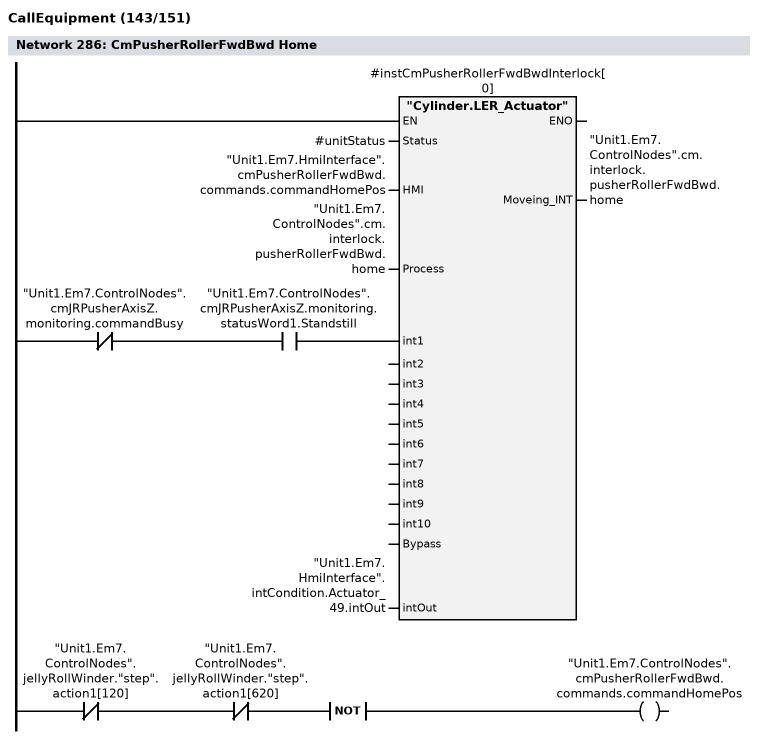
   RUNG wire#powerrail
      #instCmPusherRollerFwdBwdInterlock[0](int1 := wire#w1, Status := #unitStatus, HMI := "Unit1.Em7.HmiInterface".cmPusherRollerFwdBwd.commands.commandHomePos, Process := "Unit1.Em7.ControlNodes".cm.interlock.pusherRollerFwdBwd.home, int2 :=, int3 :=, int4 :=, int5 :=, int6 :=, int7 :=, int8 :=, int9 :=, int10 :=, Bypass :=, intOut := "Unit1.Em7.HmiInterface".intCondition.Actuator_49.intOut, Moveing_INT => "Unit1.Em7.ControlNodes".cm.interlock.pusherRollerFwdBwd.home)
   END_RUNG
   RUNG wire#powerrail
      I_Contact( "Unit1.Em7.ControlNodes".cmJRPusherAxisZ.monitoring.commandBusy )
      Contact( "Unit1.Em7.ControlNodes".cmJRPusherAxisZ.monitoring.statusWord1.Standstill )
   END_RUNG wire#w1
   RUNG wire#powerrail
      I_Contact( "Unit1.Em7.ControlNodes".jellyRollWinder."step".action1[120] )
      I_Contact( "Unit1.Em7.ControlNodes".jellyRollWinder."step".action1[620] )
      Not()
      Coil( "Unit1.Em7.ControlNodes".cmPusherRollerFwdBwd.commands.commandHomePos )
   END_RUNG
   // the same network as SCL:
   #instCmPusherRollerFwdBwdInterlock[0](Status := #unitStatus,   // "Cylinder.LER_Actuator"
                           HMI := "Unit1.Em7.HmiInterface".cmPusherRollerFwdBwd.commands.commandHomePos,
                           Process := "Unit1.Em7.ControlNodes".cm.interlock.pusherRollerFwdBwd.home,
                           int1 := NOT "Unit1.Em7.ControlNodes".cmJRPusherAxisZ.monitoring.commandBusy AND "Unit1.Em7.ControlNodes".cmJRPusherAxisZ.monitoring.statusWord1.Standstill,
                           intOut := "Unit1.Em7.HmiInterface".intCondition.Actuator_49.intOut,
                           Moveing_INT => "Unit1.Em7.ControlNodes".cm.interlock.pusherRollerFwdBwd.home);
   "Unit1.Em7.ControlNodes".cmPusherRollerFwdBwd.commands.commandHomePos := NOT (NOT "Unit1.Em7.ControlNodes".jellyRollWinder."step".action1[120] AND NOT "Unit1.Em7.ControlNodes".jellyRollWinder."step".action1[620]);
END_REGION

REGION Network 287: CmPusherRollerFwdBwd Work
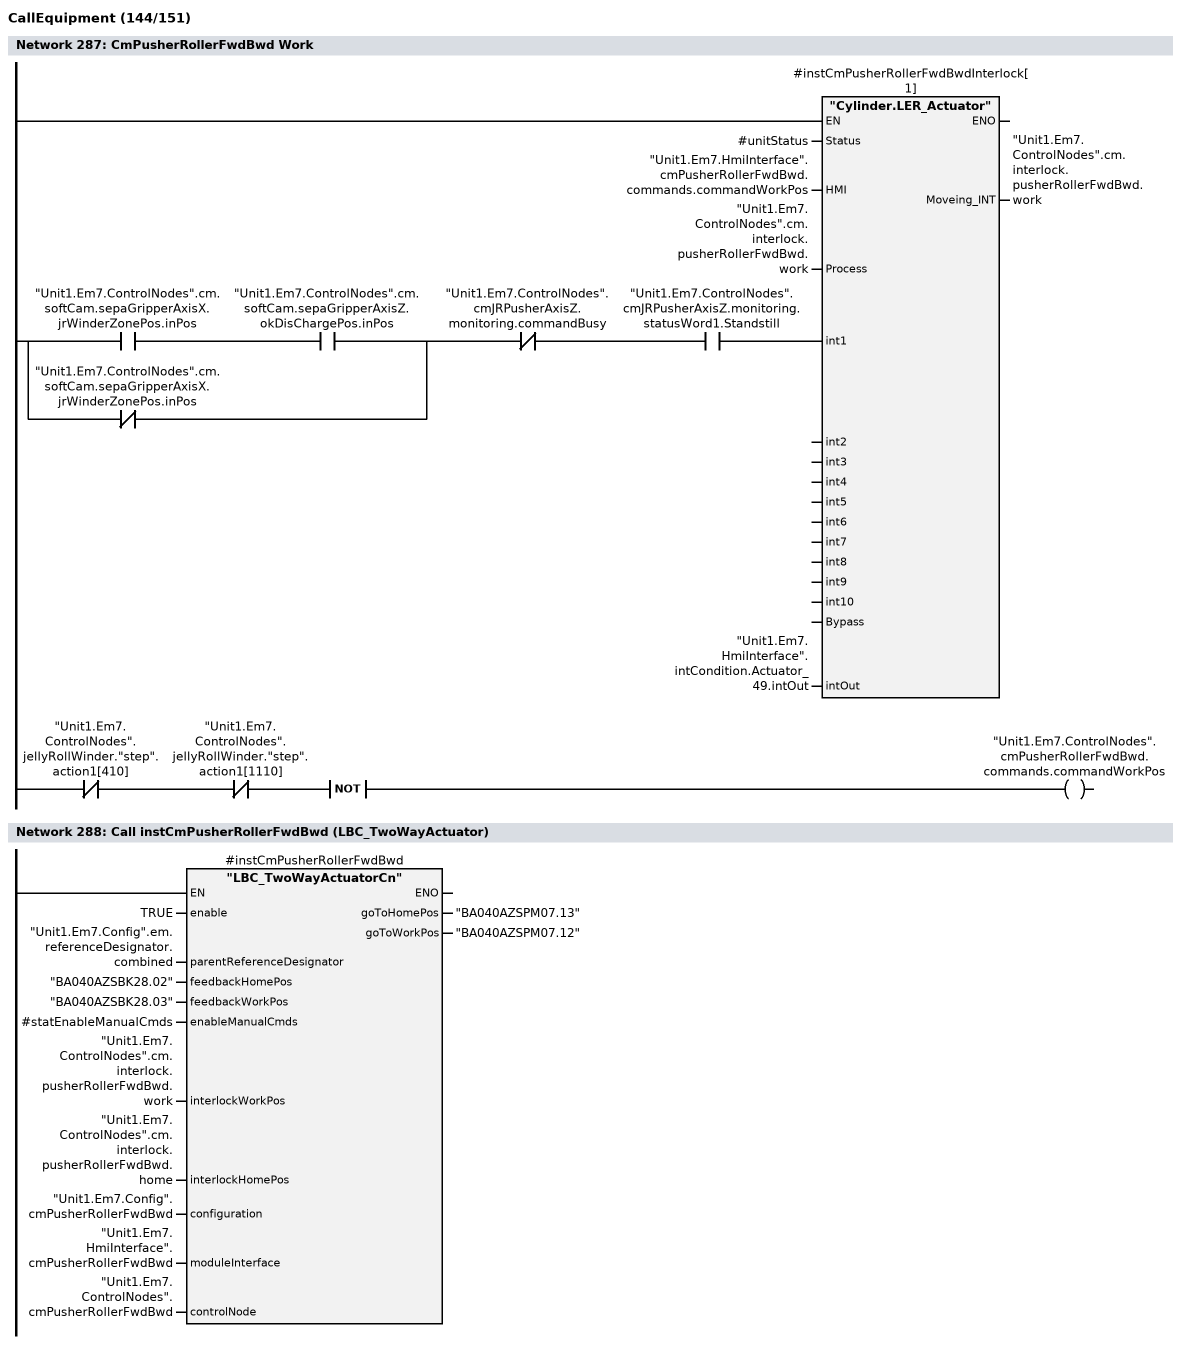
   RUNG wire#powerrail
      #instCmPusherRollerFwdBwdInterlock[1](int1 := wire#w2, Status := #unitStatus, HMI := "Unit1.Em7.HmiInterface".cmPusherRollerFwdBwd.commands.commandWorkPos, Process := "Unit1.Em7.ControlNodes".cm.interlock.pusherRollerFwdBwd.work, int2 :=, int3 :=, int4 :=, int5 :=, int6 :=, int7 :=, int8 :=, int9 :=, int10 :=, Bypass :=, intOut := "Unit1.Em7.HmiInterface".intCondition.Actuator_49.intOut, Moveing_INT => "Unit1.Em7.ControlNodes".cm.interlock.pusherRollerFwdBwd.work)
   END_RUNG
   RUNG wire#powerrail
      Contact( "Unit1.Em7.ControlNodes".cm.softCam.sepaGripperAxisX.jrWinderZonePos.inPos )
      Contact( "Unit1.Em7.ControlNodes".cm.softCam.sepaGripperAxisZ.okDisChargePos.inPos )
      wire#w1
      I_Contact( "Unit1.Em7.ControlNodes".cmJRPusherAxisZ.monitoring.commandBusy )
      Contact( "Unit1.Em7.ControlNodes".cmJRPusherAxisZ.monitoring.statusWord1.Standstill )
   END_RUNG wire#w2
   RUNG wire#powerrail
      I_Contact( "Unit1.Em7.ControlNodes".cm.softCam.sepaGripperAxisX.jrWinderZonePos.inPos )
   END_RUNG wire#w1
   RUNG wire#powerrail
      I_Contact( "Unit1.Em7.ControlNodes".jellyRollWinder."step".action1[410] )
      I_Contact( "Unit1.Em7.ControlNodes".jellyRollWinder."step".action1[1110] )
      Not()
      Coil( "Unit1.Em7.ControlNodes".cmPusherRollerFwdBwd.commands.commandWorkPos )
   END_RUNG
   // the same network as SCL:
   #instCmPusherRollerFwdBwdInterlock[1](Status := #unitStatus,   // "Cylinder.LER_Actuator"
                           HMI := "Unit1.Em7.HmiInterface".cmPusherRollerFwdBwd.commands.commandWorkPos,
                           Process := "Unit1.Em7.ControlNodes".cm.interlock.pusherRollerFwdBwd.work,
                           int1 := (("Unit1.Em7.ControlNodes".cm.softCam.sepaGripperAxisX.jrWinderZonePos.inPos AND "Unit1.Em7.ControlNodes".cm.softCam.sepaGripperAxisZ.okDisChargePos.inPos) OR NOT "Unit1.Em7.ControlNodes".cm.softCam.sepaGripperAxisX.jrWinderZonePos.inPos) AND NOT "Unit1.Em7.ControlNodes".cmJRPusherAxisZ.monitoring.commandBusy AND "Unit1.Em7.ControlNodes".cmJRPusherAxisZ.monitoring.statusWord1.Standstill,
                           intOut := "Unit1.Em7.HmiInterface".intCondition.Actuator_49.intOut,
                           Moveing_INT => "Unit1.Em7.ControlNodes".cm.interlock.pusherRollerFwdBwd.work);
   "Unit1.Em7.ControlNodes".cmPusherRollerFwdBwd.commands.commandWorkPos := NOT (NOT "Unit1.Em7.ControlNodes".jellyRollWinder."step".action1[410] AND NOT "Unit1.Em7.ControlNodes".jellyRollWinder."step".action1[1110]);
END_REGION

REGION Network 288: Call instCmPusherRollerFwdBwd (LBC_TwoWayActuator)
   RUNG wire#powerrail
      #instCmPusherRollerFwdBwd(enable := TRUE, parentReferenceDesignator := "Unit1.Em7.Config".em.referenceDesignator.combined, feedbackHomePos := "BA040AZSBK28.02", feedbackWorkPos := "BA040AZSBK28.03", enableManualCmds := #statEnableManualCmds, interlockWorkPos := "Unit1.Em7.ControlNodes".cm.interlock.pusherRollerFwdBwd.work, interlockHomePos := "Unit1.Em7.ControlNodes".cm.interlock.pusherRollerFwdBwd.home, configuration := "Unit1.Em7.Config".cmPusherRollerFwdBwd, moduleInterface := "Unit1.Em7.HmiInterface".cmPusherRollerFwdBwd, controlNode := "Unit1.Em7.ControlNodes".cmPusherRollerFwdBwd, goToHomePos => "BA040AZSPM07.13", goToWorkPos => "BA040AZSPM07.12")
   END_RUNG
   // the same network as SCL:
   #instCmPusherRollerFwdBwd(enable := TRUE,   // "LBC_TwoWayActuatorCn"
                           parentReferenceDesignator := "Unit1.Em7.Config".em.referenceDesignator.combined,
                           feedbackHomePos := "BA040AZSBK28.02",
                           feedbackWorkPos := "BA040AZSBK28.03",
                           enableManualCmds := #statEnableManualCmds,
                           interlockWorkPos := "Unit1.Em7.ControlNodes".cm.interlock.pusherRollerFwdBwd.work,
                           interlockHomePos := "Unit1.Em7.ControlNodes".cm.interlock.pusherRollerFwdBwd.home,
                           configuration := "Unit1.Em7.Config".cmPusherRollerFwdBwd,
                           moduleInterface := "Unit1.Em7.HmiInterface".cmPusherRollerFwdBwd,
                           controlNode := "Unit1.Em7.ControlNodes".cmPusherRollerFwdBwd,
                           goToHomePos => "BA040AZSPM07.13",
                           goToWorkPos => "BA040AZSPM07.12");
END_REGION

REGION Network 290: ********** Feedback to Unit **********
END_REGION

REGION Network 291: Determine StateComplete (SC) in Mode Production
   // Conditions for the Equipment Modules "stateComplete" feedback to the unit. This feedback is given when the task in for the respective state is complete.
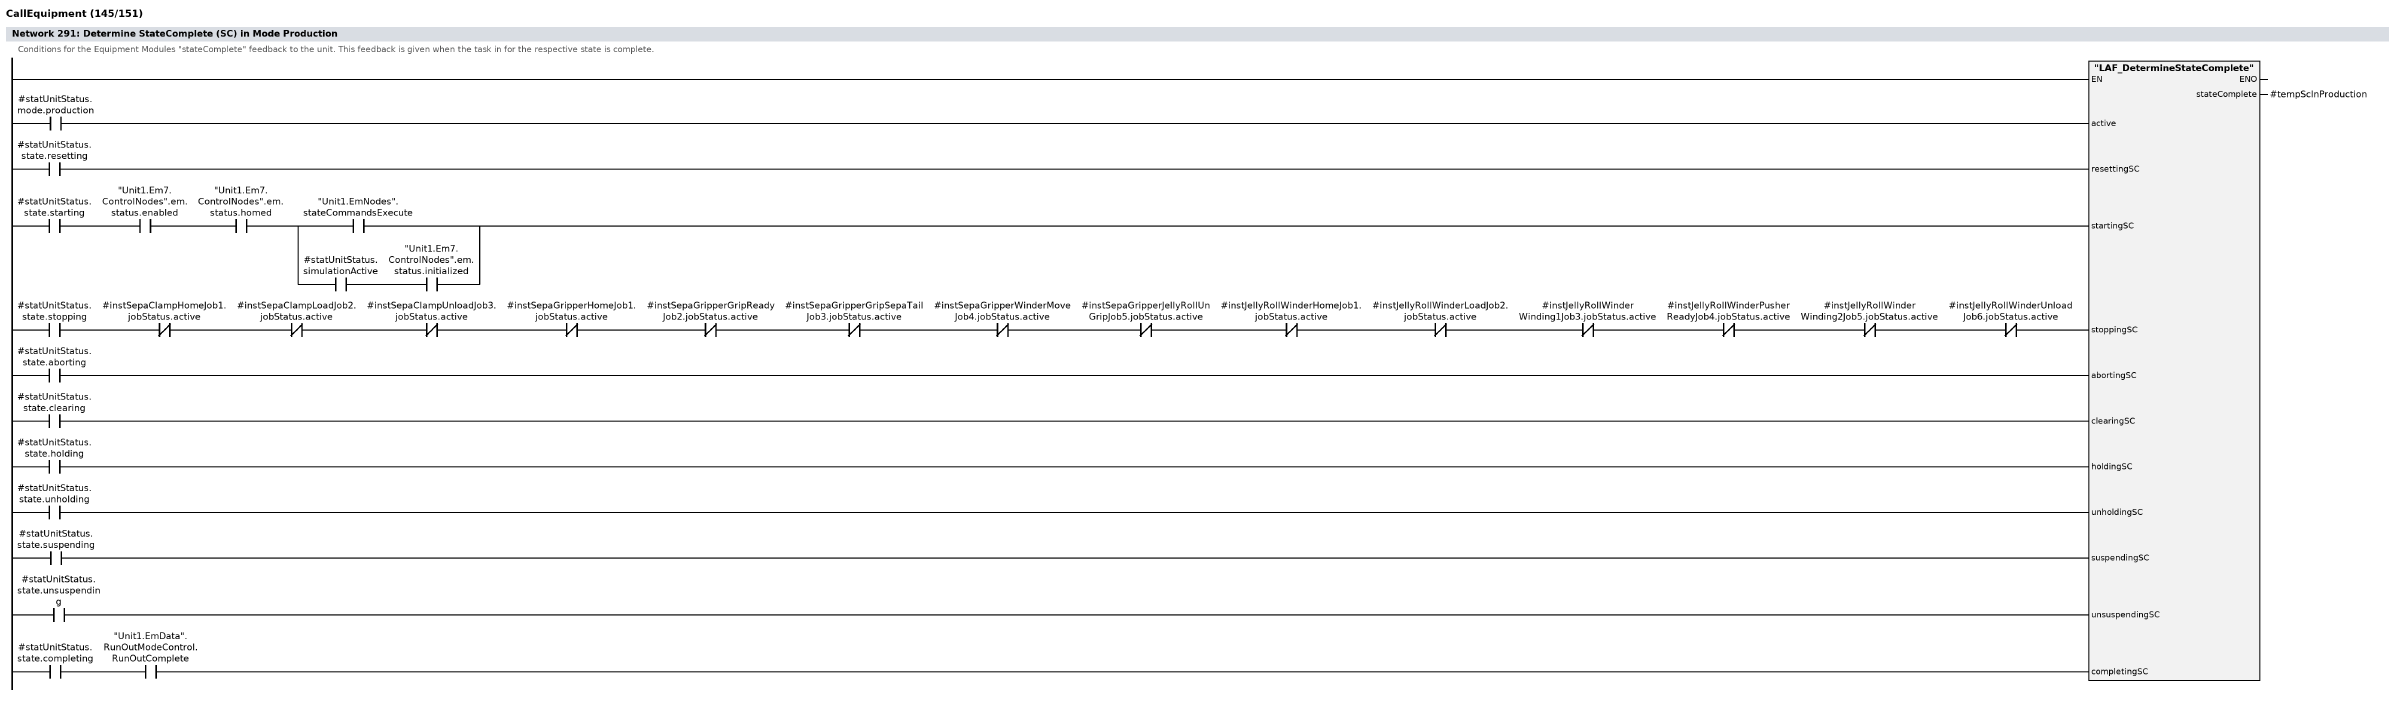
   RUNG wire#powerrail
      "LAF_DetermineStateComplete"(active := wire#w1, resettingSC := wire#w2, startingSC := wire#w4, stoppingSC := wire#w5, abortingSC := wire#w6, clearingSC := wire#w7, holdingSC := wire#w8, unholdingSC := wire#w9, suspendingSC := wire#w10, unsuspendingSC := wire#w11, completingSC := wire#w12, stateComplete => #tempScInProduction)
   END_RUNG
   RUNG wire#powerrail
      Contact( #statUnitStatus.mode.production )
   END_RUNG wire#w1
   RUNG wire#powerrail
      Contact( #statUnitStatus.state.resetting )
   END_RUNG wire#w2
   RUNG wire#powerrail
      Contact( #statUnitStatus.state.starting )
      Contact( "Unit1.Em7.ControlNodes".em.status.enabled )
      Contact( "Unit1.Em7.ControlNodes".em.status.homed )
      wire#w3
      Contact( "Unit1.EmNodes".stateCommandsExecute )
   END_RUNG wire#w4
   RUNG wire#w3
      Contact( #statUnitStatus.simulationActive )
      Contact( "Unit1.Em7.ControlNodes".em.status.initialized )
   END_RUNG wire#w4
   RUNG wire#powerrail
      Contact( #statUnitStatus.state.stopping )
      I_Contact( #instSepaClampHomeJob1.jobStatus.active )
      I_Contact( #instSepaClampLoadJob2.jobStatus.active )
      I_Contact( #instSepaClampUnloadJob3.jobStatus.active )
      I_Contact( #instSepaGripperHomeJob1.jobStatus.active )
      I_Contact( #instSepaGripperGripReadyJob2.jobStatus.active )
      I_Contact( #instSepaGripperGripSepaTailJob3.jobStatus.active )
      I_Contact( #instSepaGripperWinderMoveJob4.jobStatus.active )
      I_Contact( #instSepaGripperJellyRollUnGripJob5.jobStatus.active )
      I_Contact( #instJellyRollWinderHomeJob1.jobStatus.active )
      I_Contact( #instJellyRollWinderLoadJob2.jobStatus.active )
      I_Contact( #instJellyRollWinderWinding1Job3.jobStatus.active )
      I_Contact( #instJellyRollWinderPusherReadyJob4.jobStatus.active )
      I_Contact( #instJellyRollWinderWinding2Job5.jobStatus.active )
      I_Contact( #instJellyRollWinderUnloadJob6.jobStatus.active )
   END_RUNG wire#w5
   RUNG wire#powerrail
      Contact( #statUnitStatus.state.aborting )
   END_RUNG wire#w6
   RUNG wire#powerrail
      Contact( #statUnitStatus.state.clearing )
   END_RUNG wire#w7
   RUNG wire#powerrail
      Contact( #statUnitStatus.state.holding )
   END_RUNG wire#w8
   RUNG wire#powerrail
      Contact( #statUnitStatus.state.unholding )
   END_RUNG wire#w9
   RUNG wire#powerrail
      Contact( #statUnitStatus.state.suspending )
   END_RUNG wire#w10
   RUNG wire#powerrail
      Contact( #statUnitStatus.state.unsuspending )
   END_RUNG wire#w11
   RUNG wire#powerrail
      Contact( #statUnitStatus.state.completing )
      Contact( "Unit1.EmData".RunOutModeControl.RunOutComplete )
   END_RUNG wire#w12
   // the same network as SCL:
   "LAF_DetermineStateComplete"(active := #statUnitStatus.mode.production,
                           resettingSC := #statUnitStatus.state.resetting,
                           startingSC := #statUnitStatus.state.starting AND "Unit1.Em7.ControlNodes".em.status.enabled AND "Unit1.Em7.ControlNodes".em.status.homed AND ("Unit1.EmNodes".stateCommandsExecute OR (#statUnitStatus.simulationActive AND "Unit1.Em7.ControlNodes".em.status.initialized)),
                           stoppingSC := #statUnitStatus.state.stopping AND NOT #instSepaClampHomeJob1.jobStatus.active AND NOT #instSepaClampLoadJob2.jobStatus.active AND NOT #instSepaClampUnloadJob3.jobStatus.active AND NOT #instSepaGripperHomeJob1.jobStatus.active AND NOT #instSepaGripperGripReadyJob2.jobStatus.active AND NOT #instSepaGripperGripSepaTailJob3.jobStatus.active AND NOT #instSepaGripperWinderMoveJob4.jobStatus.active AND NOT #instSepaGripperJellyRollUnGripJob5.jobStatus.active AND NOT #instJellyRollWinderHomeJob1.jobStatus.active AND NOT #instJellyRollWinderLoadJob2.jobStatus.active AND NOT #instJellyRollWinderWinding1Job3.jobStatus.active AND NOT #instJellyRollWinderPusherReadyJob4.jobStatus.active AND NOT #instJellyRollWinderWinding2Job5.jobStatus.active AND NOT #instJellyRollWinderUnloadJob6.jobStatus.active,
                           abortingSC := #statUnitStatus.state.aborting,
                           clearingSC := #statUnitStatus.state.clearing,
                           holdingSC := #statUnitStatus.state.holding,
                           unholdingSC := #statUnitStatus.state.unholding,
                           suspendingSC := #statUnitStatus.state.suspending,
                           unsuspendingSC := #statUnitStatus.state.unsuspending,
                           completingSC := #statUnitStatus.state.completing AND "Unit1.EmData".RunOutModeControl.RunOutComplete,
                           stateComplete => #tempScInProduction);
END_REGION

REGION Network 292: Determine StateComplete (SC) in Mode Maintenance/Manual
   // Conditions for the Equipment Modules "stateComplete" feedback to the unit. This feedback is given when the task in for the respective state is complete.
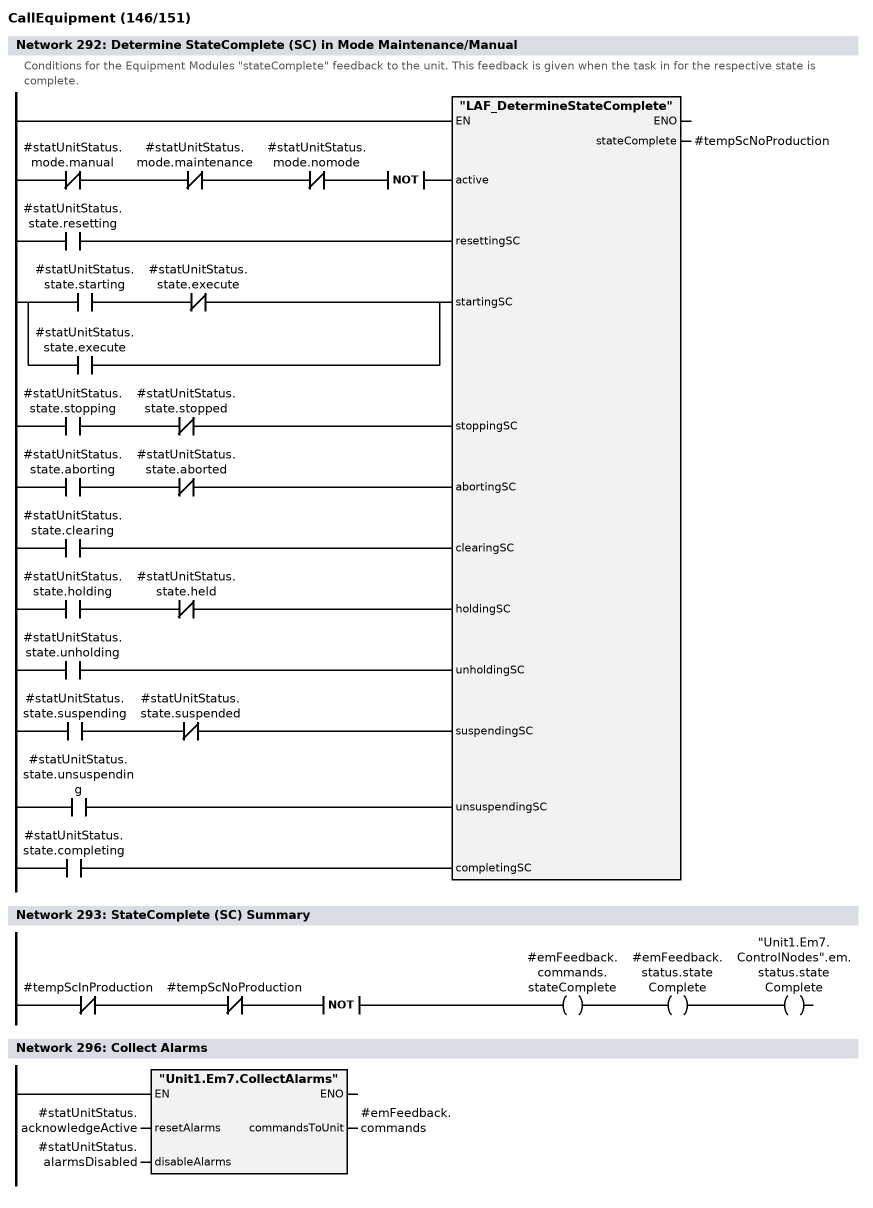
   RUNG wire#powerrail
      "LAF_DetermineStateComplete"(active := wire#w1, resettingSC := wire#w2, startingSC := wire#w3, stoppingSC := wire#w4, abortingSC := wire#w5, clearingSC := wire#w6, holdingSC := wire#w7, unholdingSC := wire#w8, suspendingSC := wire#w9, unsuspendingSC := wire#w10, completingSC := wire#w11, stateComplete => #tempScNoProduction)
   END_RUNG
   RUNG wire#powerrail
      I_Contact( #statUnitStatus.mode.manual )
      I_Contact( #statUnitStatus.mode.maintenance )
      I_Contact( #statUnitStatus.mode.nomode )
      Not()
   END_RUNG wire#w1
   RUNG wire#powerrail
      Contact( #statUnitStatus.state.resetting )
   END_RUNG wire#w2
   RUNG wire#powerrail
      Contact( #statUnitStatus.state.starting )
      I_Contact( #statUnitStatus.state.execute )
   END_RUNG wire#w3
   RUNG wire#powerrail
      Contact( #statUnitStatus.state.execute )
   END_RUNG wire#w3
   RUNG wire#powerrail
      Contact( #statUnitStatus.state.stopping )
      I_Contact( #statUnitStatus.state.stopped )
   END_RUNG wire#w4
   RUNG wire#powerrail
      Contact( #statUnitStatus.state.aborting )
      I_Contact( #statUnitStatus.state.aborted )
   END_RUNG wire#w5
   RUNG wire#powerrail
      Contact( #statUnitStatus.state.clearing )
   END_RUNG wire#w6
   RUNG wire#powerrail
      Contact( #statUnitStatus.state.holding )
      I_Contact( #statUnitStatus.state.held )
   END_RUNG wire#w7
   RUNG wire#powerrail
      Contact( #statUnitStatus.state.unholding )
   END_RUNG wire#w8
   RUNG wire#powerrail
      Contact( #statUnitStatus.state.suspending )
      I_Contact( #statUnitStatus.state.suspended )
   END_RUNG wire#w9
   RUNG wire#powerrail
      Contact( #statUnitStatus.state.unsuspending )
   END_RUNG wire#w10
   RUNG wire#powerrail
      Contact( #statUnitStatus.state.completing )
   END_RUNG wire#w11
   // the same network as SCL:
   "LAF_DetermineStateComplete"(active := NOT (NOT #statUnitStatus.mode.manual AND NOT #statUnitStatus.mode.maintenance AND NOT #statUnitStatus.mode.nomode),
                           resettingSC := #statUnitStatus.state.resetting,
                           startingSC := (#statUnitStatus.state.starting AND NOT #statUnitStatus.state.execute) OR #statUnitStatus.state.execute,
                           stoppingSC := #statUnitStatus.state.stopping AND NOT #statUnitStatus.state.stopped,
                           abortingSC := #statUnitStatus.state.aborting AND NOT #statUnitStatus.state.aborted,
                           clearingSC := #statUnitStatus.state.clearing,
                           holdingSC := #statUnitStatus.state.holding AND NOT #statUnitStatus.state.held,
                           unholdingSC := #statUnitStatus.state.unholding,
                           suspendingSC := #statUnitStatus.state.suspending AND NOT #statUnitStatus.state.suspended,
                           unsuspendingSC := #statUnitStatus.state.unsuspending,
                           completingSC := #statUnitStatus.state.completing,
                           stateComplete => #tempScNoProduction);
END_REGION

REGION Network 293: StateComplete (SC) Summary
   RUNG wire#powerrail
      I_Contact( #tempScInProduction )
      I_Contact( #tempScNoProduction )
      Not()
      Coil( #emFeedback.commands.stateComplete )
      Coil( #emFeedback.status.stateComplete )
      Coil( "Unit1.Em7.ControlNodes".em.status.stateComplete )
   END_RUNG
   // the same network as SCL:
   #emFeedback.commands.stateComplete := NOT (NOT #tempScInProduction AND NOT #tempScNoProduction);
   #emFeedback.status.stateComplete := #emFeedback.commands.stateComplete;
   "Unit1.Em7.ControlNodes".em.status.stateComplete := #emFeedback.commands.stateComplete;
END_REGION

REGION Network 295: ********** Alarms **********
END_REGION

REGION Network 296: Collect Alarms
   RUNG wire#powerrail
      "Unit1.Em7.CollectAlarms"(resetAlarms := #statUnitStatus.acknowledgeActive, disableAlarms := #statUnitStatus.alarmsDisabled, commandsToUnit => #emFeedback.commands)
   END_RUNG
   // the same network as SCL:
   "Unit1.Em7.CollectAlarms"(resetAlarms := #statUnitStatus.acknowledgeActive,
                           disableAlarms := #statUnitStatus.alarmsDisabled,
                           commandsToUnit => #emFeedback.commands);
END_REGION

REGION Network 297: Manage Alarms
   // Derive commands from the ProDiag supervision. The ProDiag supervisions contain categories which define the reaction of these supervisions (e.g. abort, stop, hold). These are handed over as commands to the unit level.
   // Alternatively, if no ProDiag should be used, you can use the LAF_ManageBitAlarms to realize bit alarm handling. This block can be found in LAF in folder 70_AlarmHandling.
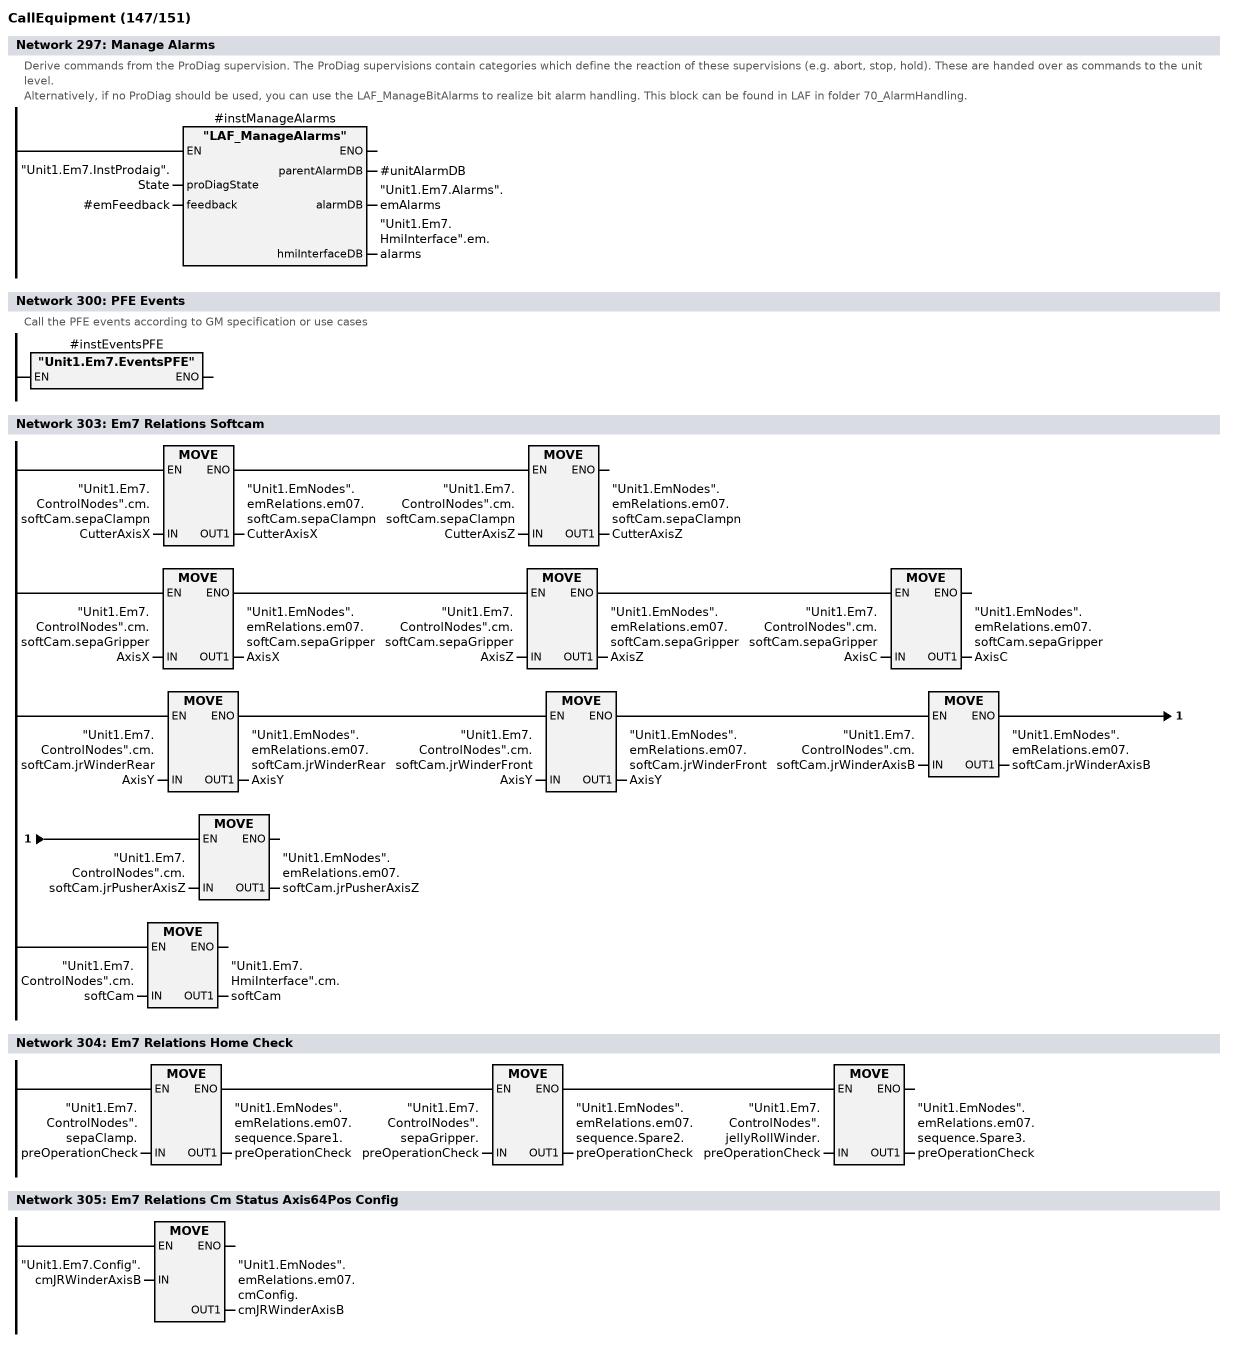
   RUNG wire#powerrail
      #instManageAlarms(proDiagState := "Unit1.Em7.InstProdaig".State, feedback := #emFeedback, parentAlarmDB => #unitAlarmDB, alarmDB => "Unit1.Em7.Alarms".emAlarms, hmiInterfaceDB => "Unit1.Em7.HmiInterface".em.alarms)
   END_RUNG
   // the same network as SCL:
   #instManageAlarms(proDiagState := "Unit1.Em7.InstProdaig".State,   // "LAF_ManageAlarms"
                     feedback := #emFeedback,
                     parentAlarmDB => #unitAlarmDB,
                     alarmDB => "Unit1.Em7.Alarms".emAlarms,
                     hmiInterfaceDB => "Unit1.Em7.HmiInterface".em.alarms);
END_REGION

REGION Network 299: ********** PFE Events **********
END_REGION

REGION Network 300: PFE Events
   // Call the PFE events according to GM specification or use cases
   RUNG wire#powerrail
      #instEventsPFE()
   END_RUNG
   // the same network as SCL:
   #instEventsPFE();   // "Unit1.Em7.EventsPFE"
END_REGION

REGION Network 302: ******************** Unit Output ********************
END_REGION

REGION Network 303: Em7 Relations Softcam
   RUNG wire#powerrail
      Move(in := "Unit1.Em7.ControlNodes".cm.softCam.sepaClampnCutterAxisX, out1 => "Unit1.EmNodes".emRelations.em07.softCam.sepaClampnCutterAxisX)
      Move(in := "Unit1.Em7.ControlNodes".cm.softCam.sepaClampnCutterAxisZ, out1 => "Unit1.EmNodes".emRelations.em07.softCam.sepaClampnCutterAxisZ)
   END_RUNG
   RUNG wire#powerrail
      Move(in := "Unit1.Em7.ControlNodes".cm.softCam.sepaGripperAxisX, out1 => "Unit1.EmNodes".emRelations.em07.softCam.sepaGripperAxisX)
      Move(in := "Unit1.Em7.ControlNodes".cm.softCam.sepaGripperAxisZ, out1 => "Unit1.EmNodes".emRelations.em07.softCam.sepaGripperAxisZ)
      Move(in := "Unit1.Em7.ControlNodes".cm.softCam.sepaGripperAxisC, out1 => "Unit1.EmNodes".emRelations.em07.softCam.sepaGripperAxisC)
   END_RUNG
   RUNG wire#powerrail
      Move(in := "Unit1.Em7.ControlNodes".cm.softCam.jrWinderRearAxisY, out1 => "Unit1.EmNodes".emRelations.em07.softCam.jrWinderRearAxisY)
      Move(in := "Unit1.Em7.ControlNodes".cm.softCam.jrWinderFrontAxisY, out1 => "Unit1.EmNodes".emRelations.em07.softCam.jrWinderFrontAxisY)
      Move(in := "Unit1.Em7.ControlNodes".cm.softCam.jrWinderAxisB, out1 => "Unit1.EmNodes".emRelations.em07.softCam.jrWinderAxisB)
      Move(in := "Unit1.Em7.ControlNodes".cm.softCam.jrPusherAxisZ, out1 => "Unit1.EmNodes".emRelations.em07.softCam.jrPusherAxisZ)
   END_RUNG
   RUNG wire#powerrail
      Move(in := "Unit1.Em7.ControlNodes".cm.softCam, out1 => "Unit1.Em7.HmiInterface".cm.softCam)
   END_RUNG
   // the same network as SCL:
   "Unit1.EmNodes".emRelations.em07.softCam.sepaClampnCutterAxisX := "Unit1.Em7.ControlNodes".cm.softCam.sepaClampnCutterAxisX;
   "Unit1.EmNodes".emRelations.em07.softCam.sepaClampnCutterAxisZ := "Unit1.Em7.ControlNodes".cm.softCam.sepaClampnCutterAxisZ;
   "Unit1.EmNodes".emRelations.em07.softCam.sepaGripperAxisX := "Unit1.Em7.ControlNodes".cm.softCam.sepaGripperAxisX;
   "Unit1.EmNodes".emRelations.em07.softCam.sepaGripperAxisZ := "Unit1.Em7.ControlNodes".cm.softCam.sepaGripperAxisZ;
   "Unit1.EmNodes".emRelations.em07.softCam.sepaGripperAxisC := "Unit1.Em7.ControlNodes".cm.softCam.sepaGripperAxisC;
   "Unit1.EmNodes".emRelations.em07.softCam.jrWinderRearAxisY := "Unit1.Em7.ControlNodes".cm.softCam.jrWinderRearAxisY;
   "Unit1.EmNodes".emRelations.em07.softCam.jrWinderFrontAxisY := "Unit1.Em7.ControlNodes".cm.softCam.jrWinderFrontAxisY;
   "Unit1.EmNodes".emRelations.em07.softCam.jrWinderAxisB := "Unit1.Em7.ControlNodes".cm.softCam.jrWinderAxisB;
   "Unit1.EmNodes".emRelations.em07.softCam.jrPusherAxisZ := "Unit1.Em7.ControlNodes".cm.softCam.jrPusherAxisZ;
   "Unit1.Em7.HmiInterface".cm.softCam := "Unit1.Em7.ControlNodes".cm.softCam;
END_REGION

REGION Network 304: Em7 Relations Home Check
   RUNG wire#powerrail
      Move(in := "Unit1.Em7.ControlNodes".sepaClamp.preOperationCheck, out1 => "Unit1.EmNodes".emRelations.em07.sequence.Spare1.preOperationCheck)
      Move(in := "Unit1.Em7.ControlNodes".sepaGripper.preOperationCheck, out1 => "Unit1.EmNodes".emRelations.em07.sequence.Spare2.preOperationCheck)
      Move(in := "Unit1.Em7.ControlNodes".jellyRollWinder.preOperationCheck, out1 => "Unit1.EmNodes".emRelations.em07.sequence.Spare3.preOperationCheck)
   END_RUNG
   // the same network as SCL:
   "Unit1.EmNodes".emRelations.em07.sequence.Spare1.preOperationCheck := "Unit1.Em7.ControlNodes".sepaClamp.preOperationCheck;
   "Unit1.EmNodes".emRelations.em07.sequence.Spare2.preOperationCheck := "Unit1.Em7.ControlNodes".sepaGripper.preOperationCheck;
   "Unit1.EmNodes".emRelations.em07.sequence.Spare3.preOperationCheck := "Unit1.Em7.ControlNodes".jellyRollWinder.preOperationCheck;
END_REGION

REGION Network 305: Em7 Relations Cm Status Axis64Pos Config
   RUNG wire#powerrail
      Move(in := "Unit1.Em7.Config".cmJRWinderAxisB, out1 => "Unit1.EmNodes".emRelations.em07.cmConfig.cmJRWinderAxisB)
   END_RUNG
   // the same network as SCL:
   "Unit1.EmNodes".emRelations.em07.cmConfig.cmJRWinderAxisB := "Unit1.Em7.Config".cmJRWinderAxisB;
END_REGION

REGION Network 306: Em7 Relations Cm Status Cylinder
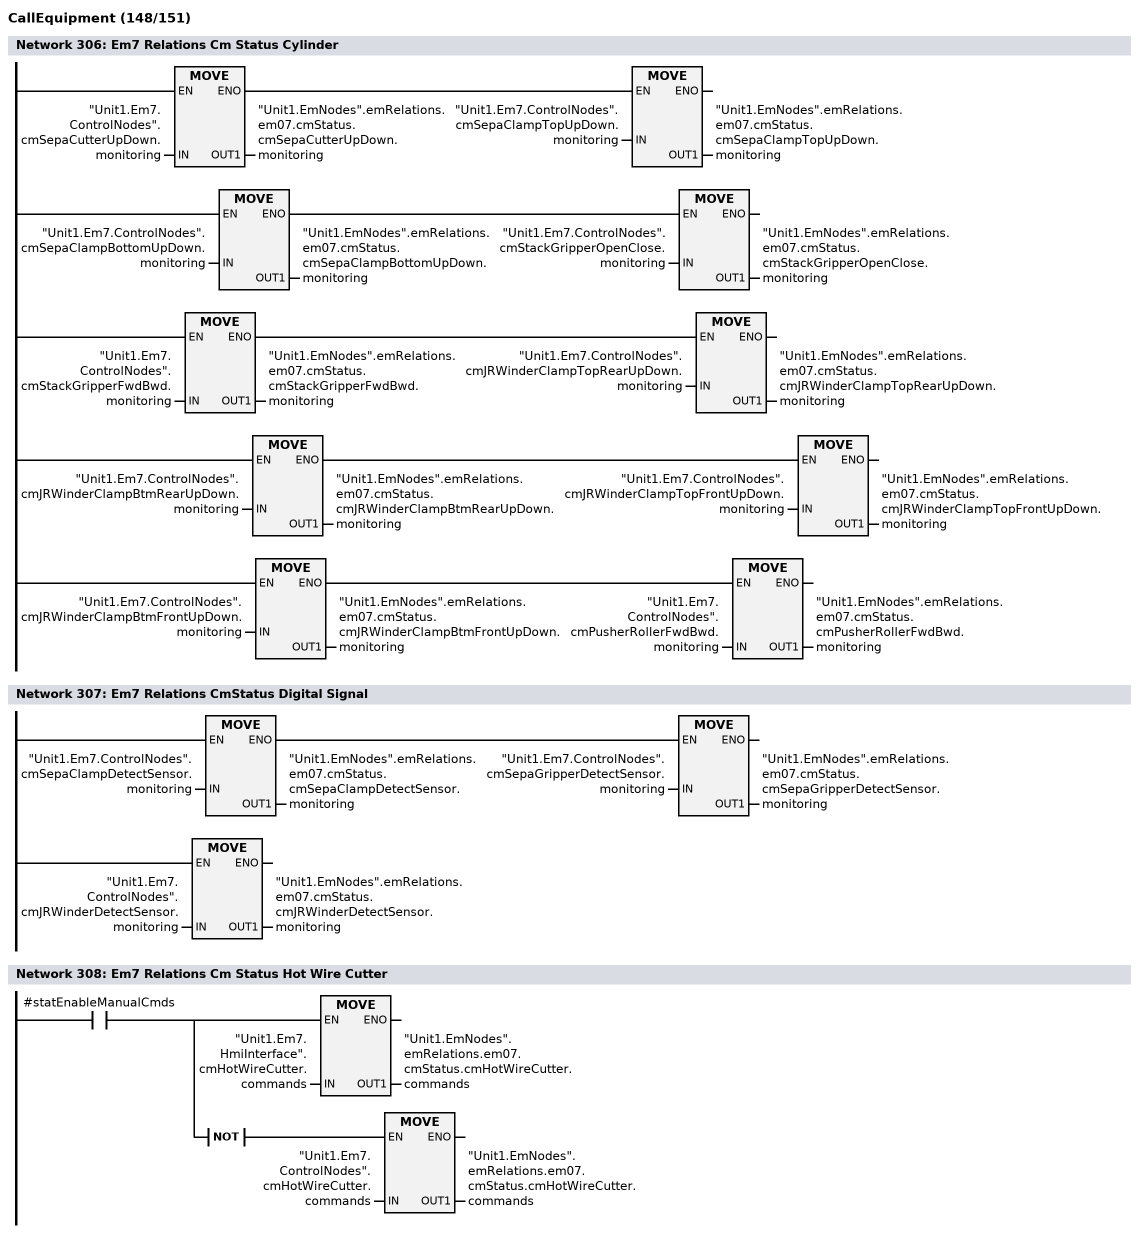
   RUNG wire#powerrail
      Move(in := "Unit1.Em7.ControlNodes".cmSepaCutterUpDown.monitoring, out1 => "Unit1.EmNodes".emRelations.em07.cmStatus.cmSepaCutterUpDown.monitoring)
      Move(in := "Unit1.Em7.ControlNodes".cmSepaClampTopUpDown.monitoring, out1 => "Unit1.EmNodes".emRelations.em07.cmStatus.cmSepaClampTopUpDown.monitoring)
   END_RUNG
   RUNG wire#powerrail
      Move(in := "Unit1.Em7.ControlNodes".cmSepaClampBottomUpDown.monitoring, out1 => "Unit1.EmNodes".emRelations.em07.cmStatus.cmSepaClampBottomUpDown.monitoring)
      Move(in := "Unit1.Em7.ControlNodes".cmStackGripperOpenClose.monitoring, out1 => "Unit1.EmNodes".emRelations.em07.cmStatus.cmStackGripperOpenClose.monitoring)
   END_RUNG
   RUNG wire#powerrail
      Move(in := "Unit1.Em7.ControlNodes".cmStackGripperFwdBwd.monitoring, out1 => "Unit1.EmNodes".emRelations.em07.cmStatus.cmStackGripperFwdBwd.monitoring)
      Move(in := "Unit1.Em7.ControlNodes".cmJRWinderClampTopRearUpDown.monitoring, out1 => "Unit1.EmNodes".emRelations.em07.cmStatus.cmJRWinderClampTopRearUpDown.monitoring)
   END_RUNG
   RUNG wire#powerrail
      Move(in := "Unit1.Em7.ControlNodes".cmJRWinderClampBtmRearUpDown.monitoring, out1 => "Unit1.EmNodes".emRelations.em07.cmStatus.cmJRWinderClampBtmRearUpDown.monitoring)
      Move(in := "Unit1.Em7.ControlNodes".cmJRWinderClampTopFrontUpDown.monitoring, out1 => "Unit1.EmNodes".emRelations.em07.cmStatus.cmJRWinderClampTopFrontUpDown.monitoring)
   END_RUNG
   RUNG wire#powerrail
      Move(in := "Unit1.Em7.ControlNodes".cmJRWinderClampBtmFrontUpDown.monitoring, out1 => "Unit1.EmNodes".emRelations.em07.cmStatus.cmJRWinderClampBtmFrontUpDown.monitoring)
      Move(in := "Unit1.Em7.ControlNodes".cmPusherRollerFwdBwd.monitoring, out1 => "Unit1.EmNodes".emRelations.em07.cmStatus.cmPusherRollerFwdBwd.monitoring)
   END_RUNG
   // the same network as SCL:
   "Unit1.EmNodes".emRelations.em07.cmStatus.cmSepaCutterUpDown.monitoring := "Unit1.Em7.ControlNodes".cmSepaCutterUpDown.monitoring;
   "Unit1.EmNodes".emRelations.em07.cmStatus.cmSepaClampTopUpDown.monitoring := "Unit1.Em7.ControlNodes".cmSepaClampTopUpDown.monitoring;
   "Unit1.EmNodes".emRelations.em07.cmStatus.cmSepaClampBottomUpDown.monitoring := "Unit1.Em7.ControlNodes".cmSepaClampBottomUpDown.monitoring;
   "Unit1.EmNodes".emRelations.em07.cmStatus.cmStackGripperOpenClose.monitoring := "Unit1.Em7.ControlNodes".cmStackGripperOpenClose.monitoring;
   "Unit1.EmNodes".emRelations.em07.cmStatus.cmStackGripperFwdBwd.monitoring := "Unit1.Em7.ControlNodes".cmStackGripperFwdBwd.monitoring;
   "Unit1.EmNodes".emRelations.em07.cmStatus.cmJRWinderClampTopRearUpDown.monitoring := "Unit1.Em7.ControlNodes".cmJRWinderClampTopRearUpDown.monitoring;
   "Unit1.EmNodes".emRelations.em07.cmStatus.cmJRWinderClampBtmRearUpDown.monitoring := "Unit1.Em7.ControlNodes".cmJRWinderClampBtmRearUpDown.monitoring;
   "Unit1.EmNodes".emRelations.em07.cmStatus.cmJRWinderClampTopFrontUpDown.monitoring := "Unit1.Em7.ControlNodes".cmJRWinderClampTopFrontUpDown.monitoring;
   "Unit1.EmNodes".emRelations.em07.cmStatus.cmJRWinderClampBtmFrontUpDown.monitoring := "Unit1.Em7.ControlNodes".cmJRWinderClampBtmFrontUpDown.monitoring;
   "Unit1.EmNodes".emRelations.em07.cmStatus.cmPusherRollerFwdBwd.monitoring := "Unit1.Em7.ControlNodes".cmPusherRollerFwdBwd.monitoring;
END_REGION

REGION Network 307: Em7 Relations CmStatus Digital Signal
   RUNG wire#powerrail
      Move(in := "Unit1.Em7.ControlNodes".cmSepaClampDetectSensor.monitoring, out1 => "Unit1.EmNodes".emRelations.em07.cmStatus.cmSepaClampDetectSensor.monitoring)
      Move(in := "Unit1.Em7.ControlNodes".cmSepaGripperDetectSensor.monitoring, out1 => "Unit1.EmNodes".emRelations.em07.cmStatus.cmSepaGripperDetectSensor.monitoring)
   END_RUNG
   RUNG wire#powerrail
      Move(in := "Unit1.Em7.ControlNodes".cmJRWinderDetectSensor.monitoring, out1 => "Unit1.EmNodes".emRelations.em07.cmStatus.cmJRWinderDetectSensor.monitoring)
   END_RUNG
   // the same network as SCL:
   "Unit1.EmNodes".emRelations.em07.cmStatus.cmSepaClampDetectSensor.monitoring := "Unit1.Em7.ControlNodes".cmSepaClampDetectSensor.monitoring;
   "Unit1.EmNodes".emRelations.em07.cmStatus.cmSepaGripperDetectSensor.monitoring := "Unit1.Em7.ControlNodes".cmSepaGripperDetectSensor.monitoring;
   "Unit1.EmNodes".emRelations.em07.cmStatus.cmJRWinderDetectSensor.monitoring := "Unit1.Em7.ControlNodes".cmJRWinderDetectSensor.monitoring;
END_REGION

REGION Network 308: Em7 Relations Cm Status Hot Wire Cutter
   RUNG wire#powerrail
      Contact( #statEnableManualCmds )
      wire#w1
      Move(in := "Unit1.Em7.HmiInterface".cmHotWireCutter.commands, out1 => "Unit1.EmNodes".emRelations.em07.cmStatus.cmHotWireCutter.commands)
   END_RUNG
   RUNG wire#w1
      Not()
      Move(in := "Unit1.Em7.ControlNodes".cmHotWireCutter.commands, out1 => "Unit1.EmNodes".emRelations.em07.cmStatus.cmHotWireCutter.commands)
   END_RUNG
   // the same network as SCL:
   IF #statEnableManualCmds THEN
       "Unit1.EmNodes".emRelations.em07.cmStatus.cmHotWireCutter.commands := "Unit1.Em7.HmiInterface".cmHotWireCutter.commands;
   END_IF;
   IF NOT #statEnableManualCmds THEN
       "Unit1.EmNodes".emRelations.em07.cmStatus.cmHotWireCutter.commands := "Unit1.Em7.ControlNodes".cmHotWireCutter.commands;
   END_IF;
END_REGION

REGION Network 309: Em7 Relations Sequence Interface
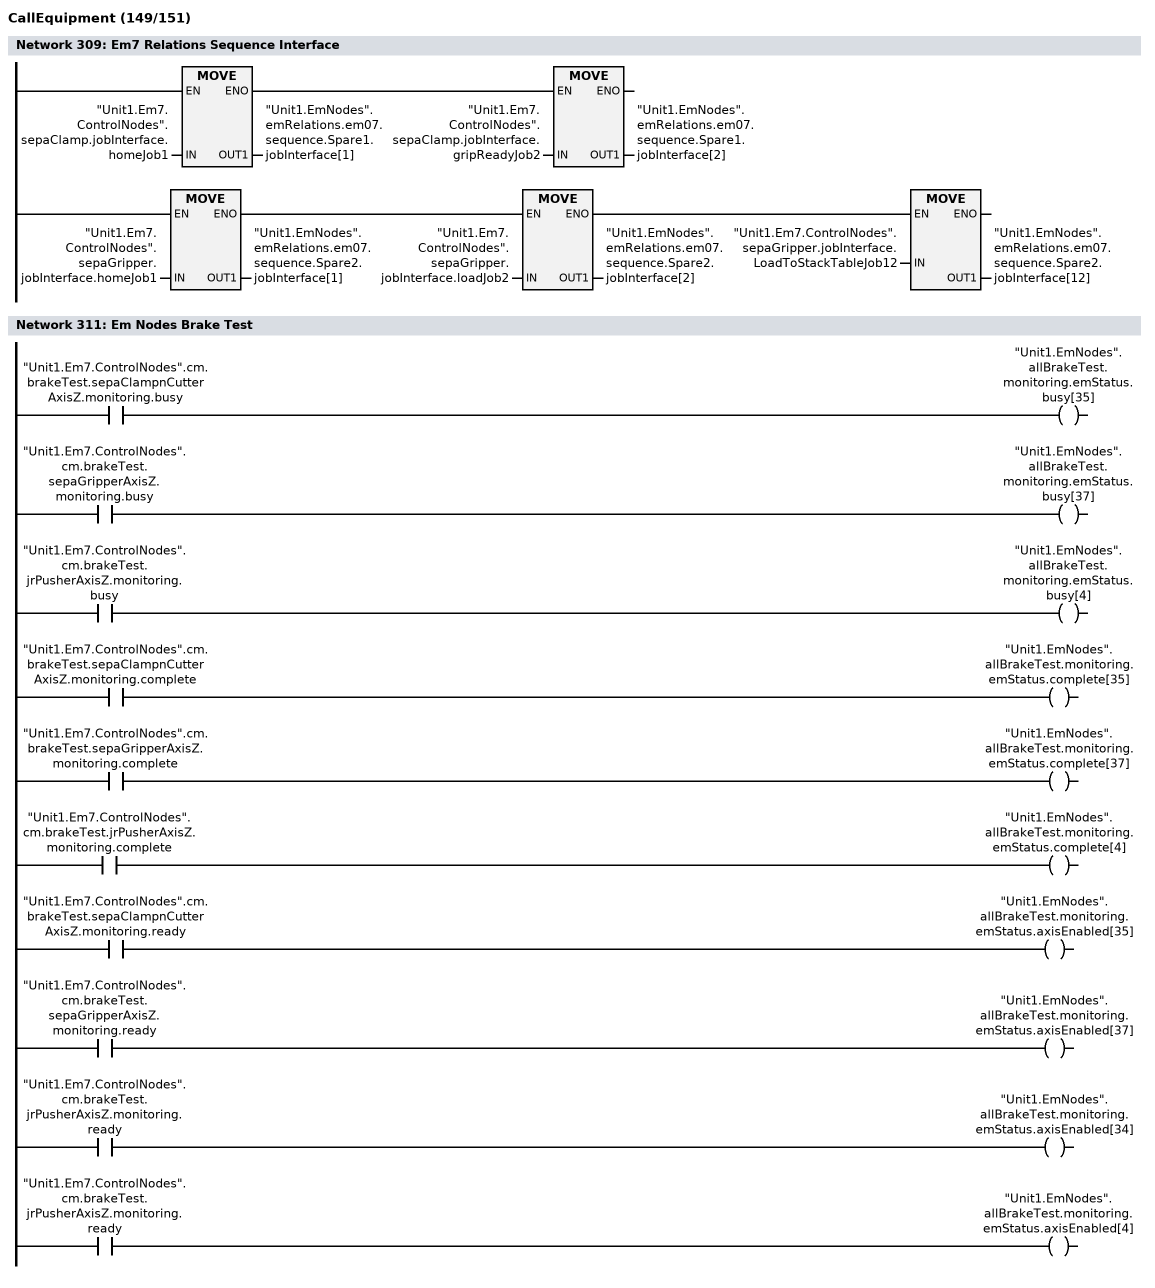
   RUNG wire#powerrail
      Move(in := "Unit1.Em7.ControlNodes".sepaClamp.jobInterface.homeJob1, out1 => "Unit1.EmNodes".emRelations.em07.sequence.Spare1.jobInterface[1])
      Move(in := "Unit1.Em7.ControlNodes".sepaClamp.jobInterface.gripReadyJob2, out1 => "Unit1.EmNodes".emRelations.em07.sequence.Spare1.jobInterface[2])
   END_RUNG
   RUNG wire#powerrail
      Move(in := "Unit1.Em7.ControlNodes".sepaGripper.jobInterface.homeJob1, out1 => "Unit1.EmNodes".emRelations.em07.sequence.Spare2.jobInterface[1])
      Move(in := "Unit1.Em7.ControlNodes".sepaGripper.jobInterface.loadJob2, out1 => "Unit1.EmNodes".emRelations.em07.sequence.Spare2.jobInterface[2])
      Move(in := "Unit1.Em7.ControlNodes".sepaGripper.jobInterface.LoadToStackTableJob12, out1 => "Unit1.EmNodes".emRelations.em07.sequence.Spare2.jobInterface[12])
   END_RUNG
   // the same network as SCL:
   "Unit1.EmNodes".emRelations.em07.sequence.Spare1.jobInterface[1] := "Unit1.Em7.ControlNodes".sepaClamp.jobInterface.homeJob1;
   "Unit1.EmNodes".emRelations.em07.sequence.Spare1.jobInterface[2] := "Unit1.Em7.ControlNodes".sepaClamp.jobInterface.gripReadyJob2;
   "Unit1.EmNodes".emRelations.em07.sequence.Spare2.jobInterface[1] := "Unit1.Em7.ControlNodes".sepaGripper.jobInterface.homeJob1;
   "Unit1.EmNodes".emRelations.em07.sequence.Spare2.jobInterface[2] := "Unit1.Em7.ControlNodes".sepaGripper.jobInterface.loadJob2;
   "Unit1.EmNodes".emRelations.em07.sequence.Spare2.jobInterface[12] := "Unit1.Em7.ControlNodes".sepaGripper.jobInterface.LoadToStackTableJob12;
END_REGION

REGION Network 310: Em Nodes BA060 Communication
END_REGION

REGION Network 311: Em Nodes Brake Test
   RUNG wire#powerrail
      Contact( "Unit1.Em7.ControlNodes".cm.brakeTest.sepaClampnCutterAxisZ.monitoring.busy )
      Coil( "Unit1.EmNodes".allBrakeTest.monitoring.emStatus.busy[35] )
   END_RUNG
   RUNG wire#powerrail
      Contact( "Unit1.Em7.ControlNodes".cm.brakeTest.sepaGripperAxisZ.monitoring.busy )
      Coil( "Unit1.EmNodes".allBrakeTest.monitoring.emStatus.busy[37] )
   END_RUNG
   RUNG wire#powerrail
      Contact( "Unit1.Em7.ControlNodes".cm.brakeTest.jrPusherAxisZ.monitoring.busy )
      Coil( "Unit1.EmNodes".allBrakeTest.monitoring.emStatus.busy[4] )
   END_RUNG
   RUNG wire#powerrail
      Contact( "Unit1.Em7.ControlNodes".cm.brakeTest.sepaClampnCutterAxisZ.monitoring.complete )
      Coil( "Unit1.EmNodes".allBrakeTest.monitoring.emStatus.complete[35] )
   END_RUNG
   RUNG wire#powerrail
      Contact( "Unit1.Em7.ControlNodes".cm.brakeTest.sepaGripperAxisZ.monitoring.complete )
      Coil( "Unit1.EmNodes".allBrakeTest.monitoring.emStatus.complete[37] )
   END_RUNG
   RUNG wire#powerrail
      Contact( "Unit1.Em7.ControlNodes".cm.brakeTest.jrPusherAxisZ.monitoring.complete )
      Coil( "Unit1.EmNodes".allBrakeTest.monitoring.emStatus.complete[4] )
   END_RUNG
   RUNG wire#powerrail
      Contact( "Unit1.Em7.ControlNodes".cm.brakeTest.sepaClampnCutterAxisZ.monitoring.ready )
      Coil( "Unit1.EmNodes".allBrakeTest.monitoring.emStatus.axisEnabled[35] )
   END_RUNG
   RUNG wire#powerrail
      Contact( "Unit1.Em7.ControlNodes".cm.brakeTest.sepaGripperAxisZ.monitoring.ready )
      Coil( "Unit1.EmNodes".allBrakeTest.monitoring.emStatus.axisEnabled[37] )
   END_RUNG
   RUNG wire#powerrail
      Contact( "Unit1.Em7.ControlNodes".cm.brakeTest.jrPusherAxisZ.monitoring.ready )
      Coil( "Unit1.EmNodes".allBrakeTest.monitoring.emStatus.axisEnabled[34] )
   END_RUNG
   RUNG wire#powerrail
      Contact( "Unit1.Em7.ControlNodes".cm.brakeTest.jrPusherAxisZ.monitoring.ready )
      Coil( "Unit1.EmNodes".allBrakeTest.monitoring.emStatus.axisEnabled[4] )
   END_RUNG
   // the same network as SCL:
   "Unit1.EmNodes".allBrakeTest.monitoring.emStatus.busy[35] := "Unit1.Em7.ControlNodes".cm.brakeTest.sepaClampnCutterAxisZ.monitoring.busy;
   "Unit1.EmNodes".allBrakeTest.monitoring.emStatus.busy[37] := "Unit1.Em7.ControlNodes".cm.brakeTest.sepaGripperAxisZ.monitoring.busy;
   "Unit1.EmNodes".allBrakeTest.monitoring.emStatus.busy[4] := "Unit1.Em7.ControlNodes".cm.brakeTest.jrPusherAxisZ.monitoring.busy;
   "Unit1.EmNodes".allBrakeTest.monitoring.emStatus.complete[35] := "Unit1.Em7.ControlNodes".cm.brakeTest.sepaClampnCutterAxisZ.monitoring.complete;
   "Unit1.EmNodes".allBrakeTest.monitoring.emStatus.complete[37] := "Unit1.Em7.ControlNodes".cm.brakeTest.sepaGripperAxisZ.monitoring.complete;
   "Unit1.EmNodes".allBrakeTest.monitoring.emStatus.complete[4] := "Unit1.Em7.ControlNodes".cm.brakeTest.jrPusherAxisZ.monitoring.complete;
   "Unit1.EmNodes".allBrakeTest.monitoring.emStatus.axisEnabled[35] := "Unit1.Em7.ControlNodes".cm.brakeTest.sepaClampnCutterAxisZ.monitoring.ready;
   "Unit1.EmNodes".allBrakeTest.monitoring.emStatus.axisEnabled[37] := "Unit1.Em7.ControlNodes".cm.brakeTest.sepaGripperAxisZ.monitoring.ready;
   "Unit1.EmNodes".allBrakeTest.monitoring.emStatus.axisEnabled[34] := "Unit1.Em7.ControlNodes".cm.brakeTest.jrPusherAxisZ.monitoring.ready;
   "Unit1.EmNodes".allBrakeTest.monitoring.emStatus.axisEnabled[4] := "Unit1.Em7.ControlNodes".cm.brakeTest.jrPusherAxisZ.monitoring.ready;
END_REGION

REGION Network 312: Homing[Temp]
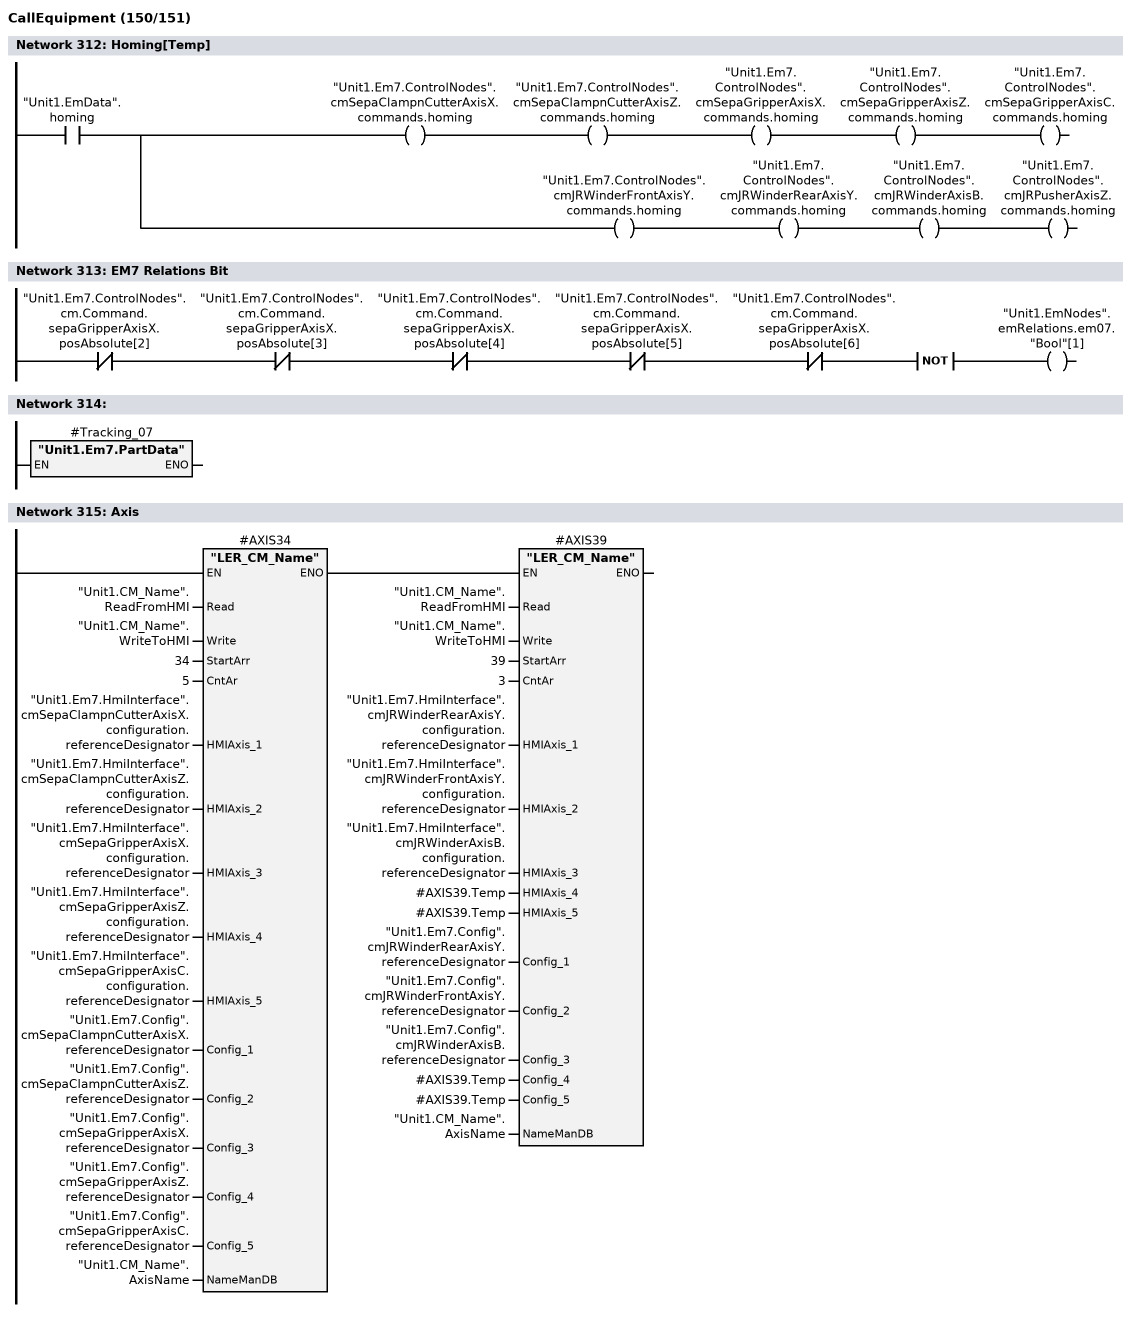
   RUNG wire#powerrail
      Contact( "Unit1.EmData".homing )
      wire#w1
      Coil( "Unit1.Em7.ControlNodes".cmSepaClampnCutterAxisX.commands.homing )
      Coil( "Unit1.Em7.ControlNodes".cmSepaClampnCutterAxisZ.commands.homing )
      Coil( "Unit1.Em7.ControlNodes".cmSepaGripperAxisX.commands.homing )
      Coil( "Unit1.Em7.ControlNodes".cmSepaGripperAxisZ.commands.homing )
      Coil( "Unit1.Em7.ControlNodes".cmSepaGripperAxisC.commands.homing )
   END_RUNG
   RUNG wire#w1
      Coil( "Unit1.Em7.ControlNodes".cmJRWinderFrontAxisY.commands.homing )
      Coil( "Unit1.Em7.ControlNodes".cmJRWinderRearAxisY.commands.homing )
      Coil( "Unit1.Em7.ControlNodes".cmJRWinderAxisB.commands.homing )
      Coil( "Unit1.Em7.ControlNodes".cmJRPusherAxisZ.commands.homing )
   END_RUNG
   // the same network as SCL:
   "Unit1.Em7.ControlNodes".cmSepaClampnCutterAxisX.commands.homing := "Unit1.EmData".homing;
   "Unit1.Em7.ControlNodes".cmSepaClampnCutterAxisZ.commands.homing := "Unit1.EmData".homing;
   "Unit1.Em7.ControlNodes".cmSepaGripperAxisX.commands.homing := "Unit1.EmData".homing;
   "Unit1.Em7.ControlNodes".cmSepaGripperAxisZ.commands.homing := "Unit1.EmData".homing;
   "Unit1.Em7.ControlNodes".cmSepaGripperAxisC.commands.homing := "Unit1.EmData".homing;
   "Unit1.Em7.ControlNodes".cmJRWinderFrontAxisY.commands.homing := "Unit1.EmData".homing;
   "Unit1.Em7.ControlNodes".cmJRWinderRearAxisY.commands.homing := "Unit1.EmData".homing;
   "Unit1.Em7.ControlNodes".cmJRWinderAxisB.commands.homing := "Unit1.EmData".homing;
   "Unit1.Em7.ControlNodes".cmJRPusherAxisZ.commands.homing := "Unit1.EmData".homing;
END_REGION

REGION Network 313: EM7 Relations Bit
   RUNG wire#powerrail
      I_Contact( "Unit1.Em7.ControlNodes".cm.Command.sepaGripperAxisX.posAbsolute[2] )
      I_Contact( "Unit1.Em7.ControlNodes".cm.Command.sepaGripperAxisX.posAbsolute[3] )
      I_Contact( "Unit1.Em7.ControlNodes".cm.Command.sepaGripperAxisX.posAbsolute[4] )
      I_Contact( "Unit1.Em7.ControlNodes".cm.Command.sepaGripperAxisX.posAbsolute[5] )
      I_Contact( "Unit1.Em7.ControlNodes".cm.Command.sepaGripperAxisX.posAbsolute[6] )
      Not()
      Coil( "Unit1.EmNodes".emRelations.em07."Bool"[1] )
   END_RUNG
   // the same network as SCL:
   "Unit1.EmNodes".emRelations.em07."Bool"[1] := NOT (NOT "Unit1.Em7.ControlNodes".cm.Command.sepaGripperAxisX.posAbsolute[2] AND NOT "Unit1.Em7.ControlNodes".cm.Command.sepaGripperAxisX.posAbsolute[3] AND NOT "Unit1.Em7.ControlNodes".cm.Command.sepaGripperAxisX.posAbsolute[4] AND NOT "Unit1.Em7.ControlNodes".cm.Command.sepaGripperAxisX.posAbsolute[5] AND NOT "Unit1.Em7.ControlNodes".cm.Command.sepaGripperAxisX.posAbsolute[6]);
END_REGION

REGION Network 314
   RUNG wire#powerrail
      #Tracking_07()
   END_RUNG
   // the same network as SCL:
   #Tracking_07();   // "Unit1.Em7.PartData"
END_REGION

REGION Network 315: Axis
   RUNG wire#powerrail
      #AXIS34(Read := "Unit1.CM_Name".ReadFromHMI, Write := "Unit1.CM_Name".WriteToHMI, StartArr := 34, CntAr := 5, HMIAxis_1 := "Unit1.Em7.HmiInterface".cmSepaClampnCutterAxisX.configuration.referenceDesignator, HMIAxis_2 := "Unit1.Em7.HmiInterface".cmSepaClampnCutterAxisZ.configuration.referenceDesignator, HMIAxis_3 := "Unit1.Em7.HmiInterface".cmSepaGripperAxisX.configuration.referenceDesignator, HMIAxis_4 := "Unit1.Em7.HmiInterface".cmSepaGripperAxisZ.configuration.referenceDesignator, HMIAxis_5 := "Unit1.Em7.HmiInterface".cmSepaGripperAxisC.configuration.referenceDesignator, Config_1 := "Unit1.Em7.Config".cmSepaClampnCutterAxisX.referenceDesignator, Config_2 := "Unit1.Em7.Config".cmSepaClampnCutterAxisZ.referenceDesignator, Config_3 := "Unit1.Em7.Config".cmSepaGripperAxisX.referenceDesignator, Config_4 := "Unit1.Em7.Config".cmSepaGripperAxisZ.referenceDesignator, Config_5 := "Unit1.Em7.Config".cmSepaGripperAxisC.referenceDesignator, NameManDB := "Unit1.CM_Name".AxisName)
      #AXIS39(Read := "Unit1.CM_Name".ReadFromHMI, Write := "Unit1.CM_Name".WriteToHMI, StartArr := 39, CntAr := 3, HMIAxis_1 := "Unit1.Em7.HmiInterface".cmJRWinderRearAxisY.configuration.referenceDesignator, HMIAxis_2 := "Unit1.Em7.HmiInterface".cmJRWinderFrontAxisY.configuration.referenceDesignator, HMIAxis_3 := "Unit1.Em7.HmiInterface".cmJRWinderAxisB.configuration.referenceDesignator, HMIAxis_4 := #AXIS39.Temp, HMIAxis_5 := #AXIS39.Temp, Config_1 := "Unit1.Em7.Config".cmJRWinderRearAxisY.referenceDesignator, Config_2 := "Unit1.Em7.Config".cmJRWinderFrontAxisY.referenceDesignator, Config_3 := "Unit1.Em7.Config".cmJRWinderAxisB.referenceDesignator, Config_4 := #AXIS39.Temp, Config_5 := #AXIS39.Temp, NameManDB := "Unit1.CM_Name".AxisName)
   END_RUNG
   // the same network as SCL:
   #AXIS34(Read := "Unit1.CM_Name".ReadFromHMI,   // "LER_CM_Name"
           Write := "Unit1.CM_Name".WriteToHMI,
           StartArr := 34,
           CntAr := 5,
           HMIAxis_1 := "Unit1.Em7.HmiInterface".cmSepaClampnCutterAxisX.configuration.referenceDesignator,
           HMIAxis_2 := "Unit1.Em7.HmiInterface".cmSepaClampnCutterAxisZ.configuration.referenceDesignator,
           HMIAxis_3 := "Unit1.Em7.HmiInterface".cmSepaGripperAxisX.configuration.referenceDesignator,
           HMIAxis_4 := "Unit1.Em7.HmiInterface".cmSepaGripperAxisZ.configuration.referenceDesignator,
           HMIAxis_5 := "Unit1.Em7.HmiInterface".cmSepaGripperAxisC.configuration.referenceDesignator,
           Config_1 := "Unit1.Em7.Config".cmSepaClampnCutterAxisX.referenceDesignator,
           Config_2 := "Unit1.Em7.Config".cmSepaClampnCutterAxisZ.referenceDesignator,
           Config_3 := "Unit1.Em7.Config".cmSepaGripperAxisX.referenceDesignator,
           Config_4 := "Unit1.Em7.Config".cmSepaGripperAxisZ.referenceDesignator,
           Config_5 := "Unit1.Em7.Config".cmSepaGripperAxisC.referenceDesignator,
           NameManDB := "Unit1.CM_Name".AxisName,
           ENO => #_w1);
   IF #_w1 THEN
       #AXIS39(Read := "Unit1.CM_Name".ReadFromHMI,   // "LER_CM_Name"
               Write := "Unit1.CM_Name".WriteToHMI,
               StartArr := 39,
               CntAr := 3,
               HMIAxis_1 := "Unit1.Em7.HmiInterface".cmJRWinderRearAxisY.configuration.referenceDesignator,
               HMIAxis_2 := "Unit1.Em7.HmiInterface".cmJRWinderFrontAxisY.configuration.referenceDesignator,
               HMIAxis_3 := "Unit1.Em7.HmiInterface".cmJRWinderAxisB.configuration.referenceDesignator,
               HMIAxis_4 := #AXIS39.Temp,
               HMIAxis_5 := #AXIS39.Temp,
               Config_1 := "Unit1.Em7.Config".cmJRWinderRearAxisY.referenceDesignator,
               Config_2 := "Unit1.Em7.Config".cmJRWinderFrontAxisY.referenceDesignator,
               Config_3 := "Unit1.Em7.Config".cmJRWinderAxisB.referenceDesignator,
               Config_4 := #AXIS39.Temp,
               Config_5 := #AXIS39.Temp,
               NameManDB := "Unit1.CM_Name".AxisName);
   END_IF;
END_REGION

REGION Network 316: Cylinder
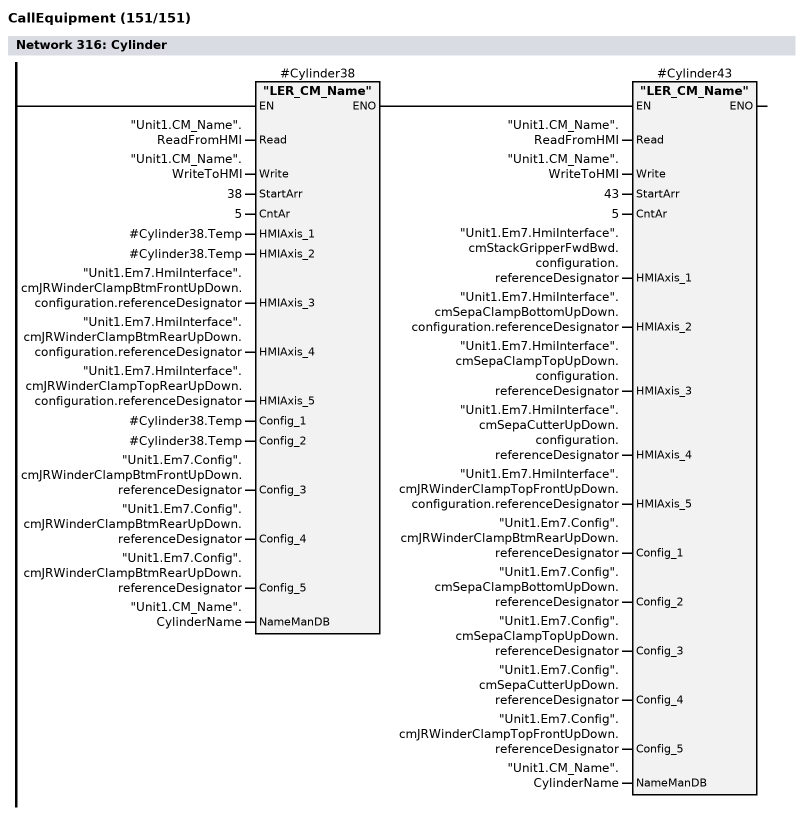
   RUNG wire#powerrail
      #Cylinder38(Read := "Unit1.CM_Name".ReadFromHMI, Write := "Unit1.CM_Name".WriteToHMI, StartArr := 38, CntAr := 5, HMIAxis_1 := #Cylinder38.Temp, HMIAxis_2 := #Cylinder38.Temp, HMIAxis_3 := "Unit1.Em7.HmiInterface".cmJRWinderClampBtmFrontUpDown.configuration.referenceDesignator, HMIAxis_4 := "Unit1.Em7.HmiInterface".cmJRWinderClampBtmRearUpDown.configuration.referenceDesignator, HMIAxis_5 := "Unit1.Em7.HmiInterface".cmJRWinderClampTopRearUpDown.configuration.referenceDesignator, Config_1 := #Cylinder38.Temp, Config_2 := #Cylinder38.Temp, Config_3 := "Unit1.Em7.Config".cmJRWinderClampBtmFrontUpDown.referenceDesignator, Config_4 := "Unit1.Em7.Config".cmJRWinderClampBtmRearUpDown.referenceDesignator, Config_5 := "Unit1.Em7.Config".cmJRWinderClampBtmRearUpDown.referenceDesignator, NameManDB := "Unit1.CM_Name".CylinderName)
      #Cylinder43(Read := "Unit1.CM_Name".ReadFromHMI, Write := "Unit1.CM_Name".WriteToHMI, StartArr := 43, CntAr := 5, HMIAxis_1 := "Unit1.Em7.HmiInterface".cmStackGripperFwdBwd.configuration.referenceDesignator, HMIAxis_2 := "Unit1.Em7.HmiInterface".cmSepaClampBottomUpDown.configuration.referenceDesignator, HMIAxis_3 := "Unit1.Em7.HmiInterface".cmSepaClampTopUpDown.configuration.referenceDesignator, HMIAxis_4 := "Unit1.Em7.HmiInterface".cmSepaCutterUpDown.configuration.referenceDesignator, HMIAxis_5 := "Unit1.Em7.HmiInterface".cmJRWinderClampTopFrontUpDown.configuration.referenceDesignator, Config_1 := "Unit1.Em7.Config".cmJRWinderClampBtmRearUpDown.referenceDesignator, Config_2 := "Unit1.Em7.Config".cmSepaClampBottomUpDown.referenceDesignator, Config_3 := "Unit1.Em7.Config".cmSepaClampTopUpDown.referenceDesignator, Config_4 := "Unit1.Em7.Config".cmSepaCutterUpDown.referenceDesignator, Config_5 := "Unit1.Em7.Config".cmJRWinderClampTopFrontUpDown.referenceDesignator, NameManDB := "Unit1.CM_Name".CylinderName)
   END_RUNG
   // the same network as SCL:
   #Cylinder38(Read := "Unit1.CM_Name".ReadFromHMI,   // "LER_CM_Name"
               Write := "Unit1.CM_Name".WriteToHMI,
               StartArr := 38,
               CntAr := 5,
               HMIAxis_1 := #Cylinder38.Temp,
               HMIAxis_2 := #Cylinder38.Temp,
               HMIAxis_3 := "Unit1.Em7.HmiInterface".cmJRWinderClampBtmFrontUpDown.configuration.referenceDesignator,
               HMIAxis_4 := "Unit1.Em7.HmiInterface".cmJRWinderClampBtmRearUpDown.configuration.referenceDesignator,
               HMIAxis_5 := "Unit1.Em7.HmiInterface".cmJRWinderClampTopRearUpDown.configuration.referenceDesignator,
               Config_1 := #Cylinder38.Temp,
               Config_2 := #Cylinder38.Temp,
               Config_3 := "Unit1.Em7.Config".cmJRWinderClampBtmFrontUpDown.referenceDesignator,
               Config_4 := "Unit1.Em7.Config".cmJRWinderClampBtmRearUpDown.referenceDesignator,
               Config_5 := "Unit1.Em7.Config".cmJRWinderClampBtmRearUpDown.referenceDesignator,
               NameManDB := "Unit1.CM_Name".CylinderName,
               ENO => #_w1);
   IF #_w1 THEN
       #Cylinder43(Read := "Unit1.CM_Name".ReadFromHMI,   // "LER_CM_Name"
                   Write := "Unit1.CM_Name".WriteToHMI,
                   StartArr := 43,
                   CntAr := 5,
                   HMIAxis_1 := "Unit1.Em7.HmiInterface".cmStackGripperFwdBwd.configuration.referenceDesignator,
                   HMIAxis_2 := "Unit1.Em7.HmiInterface".cmSepaClampBottomUpDown.configuration.referenceDesignator,
                   HMIAxis_3 := "Unit1.Em7.HmiInterface".cmSepaClampTopUpDown.configuration.referenceDesignator,
                   HMIAxis_4 := "Unit1.Em7.HmiInterface".cmSepaCutterUpDown.configuration.referenceDesignator,
                   HMIAxis_5 := "Unit1.Em7.HmiInterface".cmJRWinderClampTopFrontUpDown.configuration.referenceDesignator,
                   Config_1 := "Unit1.Em7.Config".cmJRWinderClampBtmRearUpDown.referenceDesignator,
                   Config_2 := "Unit1.Em7.Config".cmSepaClampBottomUpDown.referenceDesignator,
                   Config_3 := "Unit1.Em7.Config".cmSepaClampTopUpDown.referenceDesignator,
                   Config_4 := "Unit1.Em7.Config".cmSepaCutterUpDown.referenceDesignator,
                   Config_5 := "Unit1.Em7.Config".cmJRWinderClampTopFrontUpDown.referenceDesignator,
                   NameManDB := "Unit1.CM_Name".CylinderName);
   END_IF;
END_REGION
END_FUNCTION_BLOCK
